Fanuc KAREL source: compact_preamble.KL

PROGRAM KD00008
%TPMOTION
%NOLOCKGROUP
VAR
I:INTEGER;J:INTEGER;B:BOOLEAN;R:REAL;S : STRING[80]
BEGIN
I=1
END KD00008
